RoboDK station: Example 1 - Basic Pick and Place.rdk

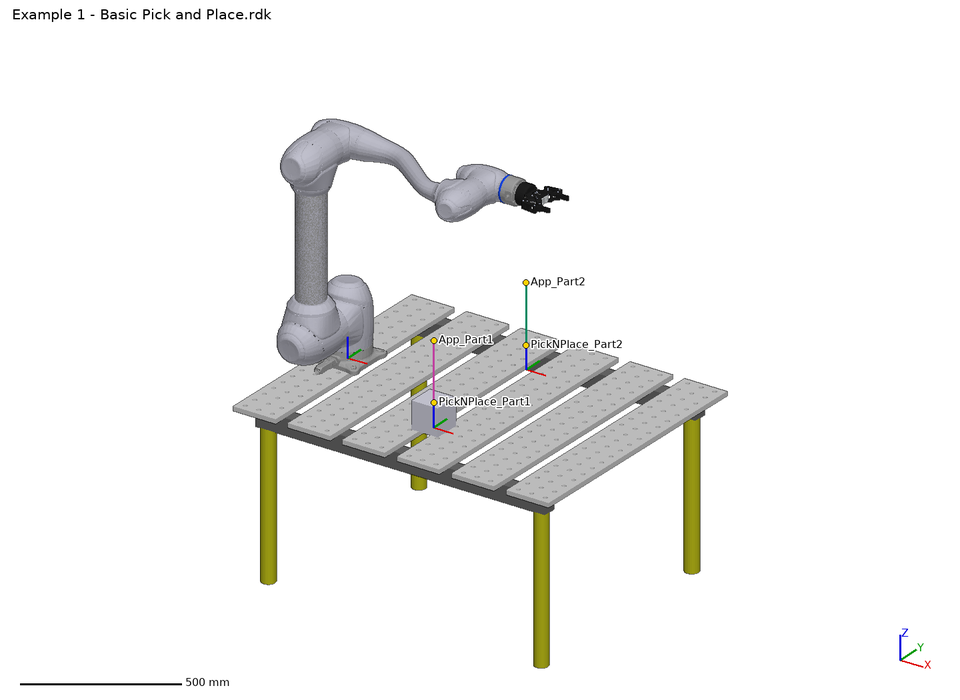
[picture v0: the station drawn from its stored meshes, robots at their saved joint values, targets as dots, program paths as lines]
Station Example 1 - Basic Pick and Place. Poses are relative to the parent item; angles as X-Y-Z fixed-axis rotations.
  - frame Doosan Robotics M1013 Base at (0, 0, 0) mm
    - robot Doosan Robotics M1013: 6 axes, payload 10 kg, reach 1300 mm, repeatability 0.1 mm, weight 33 kg
        modified DH rows (alpha deg, a mm, theta deg, d mm): 0, 0, 0, 152.5; -90, 0, -90, 34.506; 0, 620, -90, 0; -90, 0, 0, 559; 90, 0, 0, 0; -90, 0, 180, 121
        base shift (0, 0, 0) mm, rotated rx 0 ry 0 rz 180 deg
        joint limits [-360, -360, -160, -360, -360, -360] to [360, 360, 160, 360, 360, 360]; home [0, 0, -90, 0, 0, 0]; saved at [0, 0, -90, 0, 0, 0]
      - tool Gripper RobotiQ 85 Opened, TCP at (0, 0, 130) mm, size 147.4 x 146.8 x 75 mm
  - frame World at (0, 0, 0) mm
    - object Table at (500, 0, 0) mm, size 1193.8 x 965.2 x 609.6 mm, geometry from welding_table.sld
  - frame Part1 at (500, -250, 0) mm
    - target PickNPlace_Part1 (Cartesian target) at (0, 0, 85) mm, rotated rx 180 ry 0 rz 90 deg; joints [-20.504, -21.289, -113.554, 0, -45.157, -20.504] of Doosan Robotics M1013
    - target App_Part1 (Cartesian target) at (0, 0, 300) mm, rotated rx 180 ry 0 rz 90 deg; joints [-20.504, -9.701, -102.656, 0, -67.643, -20.504] of Doosan Robotics M1013
    - object box at (0, 0, 50) mm, size 100 x 100 x 100 mm, geometry from box.sld
  - frame Part2 at (500, 250, 0) mm
    - target App_Part2 (Cartesian target) at (0, 0, 300) mm, rotated rx 180 ry 0 rz 90 deg; joints [26.86, -9.701, -102.656, 0, -67.643, 26.86] of Doosan Robotics M1013
    - target PickNPlace_Part2 (Cartesian target) at (0, 0, 85) mm, rotated rx 180 ry 0 rz 90 deg; joints [26.86, -21.289, -113.554, 0, -45.157, 26.86] of Doosan Robotics M1013
  - program ReplaceObjects (1 instructions, listed below)
  - program PickPart1 (6 instructions, listed below)
  - program PlacePart2 (6 instructions, listed below)
  - program PickPart2 (6 instructions, listed below)
  - program PlacePart1 (6 instructions, listed below)
  - program MainProgram (4 instructions, listed below)
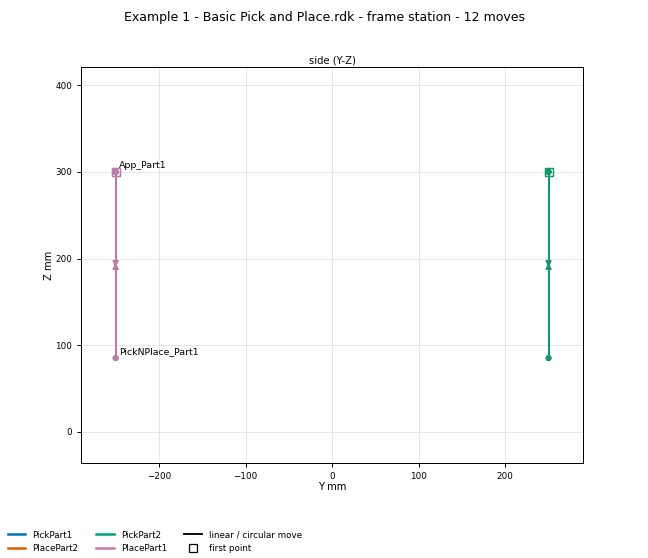
[picture p0: tool path of Example 1 - Basic Pick and Place.rdk in frame station, 12 of 12 moves have a stored position in this frame; points joined in program order, loops and branches not executed]

--- program ReplaceObjects (robot Doosan Robotics M1013) ---
  Replace objects

--- program PickPart1 (robot Doosan Robotics M1013) ---
  Set Ref.: Part1
  Set Tool: Gripper RobotiQ 85 Opened
  MoveJ (App_Part1)
  MoveL (PickNPlace_Part1)
  Attach to Gripper RobotiQ 85 Opened
  MoveL (App_Part1)

--- program PlacePart2 (robot Doosan Robotics M1013) ---
  Set Ref.: Part2
  Set Tool: Gripper RobotiQ 85 Opened
  MoveJ (App_Part2)
  MoveL (PickNPlace_Part2)
  Detach from Gripper RobotiQ 85 Opened
  MoveL (App_Part2)

--- program PickPart2 (robot Doosan Robotics M1013) ---
  Set Ref.: Part2
  Set Tool: Gripper RobotiQ 85 Opened
  MoveJ (App_Part2)
  MoveL (PickNPlace_Part2)
  Attach to Gripper RobotiQ 85 Opened
  MoveL (App_Part2)

--- program PlacePart1 (robot Doosan Robotics M1013) ---
  Set Ref.: Part1
  Set Tool: Gripper RobotiQ 85 Opened
  MoveJ (App_Part1)
  MoveL (PickNPlace_Part1)
  Detach from Gripper RobotiQ 85 Opened
  MoveL (App_Part1)

--- program MainProgram (robot Doosan Robotics M1013) ---
  Call PickPart1
  Call PlacePart2
  Call PickPart2
  Call PlacePart1
